// Some object that only implements a user defined logic.
FUNCTION_BLOCK FB_UDef_Obj EXTENDS FB_BA_Object
VAR_OUTPUT
	nCounter		: UDINT;
END_VAR

SUPER^();

nCounter := (nCounter + 1);

END_FUNCTION_BLOCK

(* stored: Version 1.1.0.1, ProductVersion 3.1.4024.9
   POU FB_UDef_Obj: Id {d154ff6f-0fbc-4d1e-9fce-7c756b18f436}, SpecialFunc None *)
